FUNCTION_BLOCK PosDeltaHighPrecRapidUpd (* The "Position Delta, High Precision Rapid Update" Parameter Group is intended for applications where very high precision and very fast update rates are needed for position data. This PGN can provide delta position changes down to 1 millimeter with a delta time period accurate to 5 milliseconds *)
  (* Standard: NMEA 2000; Classification: PGN 129027; Function: Position Delta, High Precision Rapid Update; Description: Copyright (c) 2024 HR Agrartechnik GmbH This program and the accompanying materials are made available under the terms of the Eclipse Public License 2.0 which is available at https://www.eclipse.org/legal/epl-2.0/ SPDX-License-Identifier: EPL-2.0 *)
  (* Version 1.0, 07.02.2025, Moritz Ortmeier, HR Agrartechnik GmbH *)
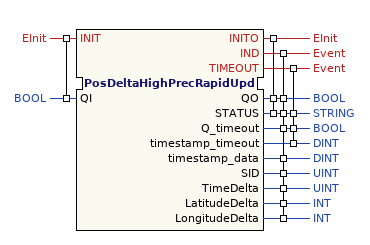
  EVENT_INPUT
    INIT : EInit WITH QI; (* Service Initialization *)
  END_EVENT
  EVENT_OUTPUT
    INITO : EInit WITH QO, STATUS; (* Initialization Confirm *)
    IND WITH QO, timestamp_data, SID, TimeDelta, LatitudeDelta, STATUS, Q_timeout, LongitudeDelta; (* Indication from Resource *)
    TIMEOUT WITH timestamp_timeout, STATUS, Q_timeout;
  END_EVENT
  VAR_INPUT
    QI : BOOL; (* Event Input Qualifier *)
  END_VAR
  VAR_OUTPUT
    QO : BOOL; (* Event Output Qualifier *)
    STATUS : STRING;
    Q_timeout : BOOL;
    timestamp_timeout : DINT;
    timestamp_data : DINT;
    SID : UINT; (* Sequence ID identifies the sequence this data is associated with so that the data can be synchronized with other vessel data for this same sequence being sent in another PGN. *)
    TimeDelta : UINT;
    LatitudeDelta : INT;
    LongitudeDelta : INT;
  END_VAR
END_FUNCTION_BLOCK
